TYPE RecipeData :
STRUCT
	fTemperature        : REAL;
	nAgitatorSpeed      : DINT;
	nMixTimeSecs        : DINT;	
END_STRUCT
END_TYPE

(* stored: Version 1.1.0.1
   DUT RecipeData: Id {6f664184-508e-4a4d-bab1-789bc21fb165} *)
